FUNCTION F_ClampReal (* Clamp a REAL value into [rMin, rMax] with over/under flags. *)
  (* Standard: 61499-2; Description: Copyright (c) 2026 Meisterschulen am Ostbahnhof This program and the accompanying materials are made available under the terms of the Eclipse Public License 2.0 which is available at https://www.eclipse.org/legal/epl-2.0/ SPDX-License-Identifier: EPL-2.0 *)
  (* Version 1.0, 2026-09-05, Franz Höpfinger, Meisterschulen am Ostbahnhof, initial API and implementation and/or initial documentation *)
  PACKAGE logiBUS::signalprocessing::clamp;
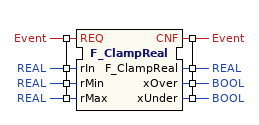
  EVENT_INPUT
    REQ WITH rIn, rMin, rMax;
  END_EVENT
  EVENT_OUTPUT
    CNF WITH F_ClampReal, xOver, xUnder;
  END_EVENT
  VAR_INPUT
    rIn : REAL;
    rMin : REAL;
    rMax : REAL;
  END_VAR
  VAR_OUTPUT
    F_ClampReal : REAL;
    xOver : BOOL;
    xUnder : BOOL;
  END_VAR
  BODY IN ST:
PACKAGE logiBUS::signalprocessing::clamp;

(* Clamp a REAL value into [rMin, rMax] with over/under flags. *)
FUNCTION F_ClampReal : REAL

VAR_INPUT
	rIn : REAL;
	rMin : REAL;
	rMax : REAL;
END_VAR

VAR_OUTPUT
	xOver : BOOL;
	xUnder : BOOL;
END_VAR

IF rIn > rMax THEN
	F_ClampReal := rMax;
	xOver := TRUE;
	xUnder := FALSE;
ELSIF rIn < rMin THEN
	F_ClampReal := rMin;
	xOver := FALSE;
	xUnder := TRUE;
ELSE
	F_ClampReal := rIn;
	xOver := FALSE;
	xUnder := FALSE;
END_IF;

END_FUNCTION
  END_BODY
END_FUNCTION
